// Mitsubishi GX Works2 project: TappingM6   PLC: FX1N/FX1NC

// global labels: Global1
VAR_GLOBAL
  XXFeed AT D52 : INT;
  XXRun AT M51 : BOOL;
  XXTarget AT D51 : INT;
  XXCurrent AT D50 : INT;
  XXArray AT D53 : ARRAY [0..5] OF INT;
  Foil3 AT M20 : BOOL;
  Foil4 AT M21 : BOOL;
  XXIMin AT X000 : BOOL;
  ZZIMin AT X001 : BOOL;
  ZZIMax AT X002 : BOOL;
  FoilExtractorIMax AT X003 : BOOL;
  XXODirection AT Y004 : BOOL;
  XXOPulse AT Y000 : BOOL;
  ZZOPulse AT Y001 : BOOL;
  RunStop AT M24 : BOOL;
  RunTest AT M23 : BOOL;
  FoilBlocker AT M54 : BOOL;
  FoilExtractor AT M55 : BOOL;
  RunState AT D20 : INT;
  Run AT M22 : BOOL;
  XXCurrentPulse AT D8140 : DINT;
  Foil3Array AT D200 : ARRAY [0..5] OF INT;
  Foil4Array AT D210 : ARRAY [0..5] OF INT;
  FoilIndex AT D70 : INT;
  RunIsTest AT M25 : BOOL;
  RunFeedXX AT D21 : INT;
  TestSensorFoil AT M30 : BOOL;
  FoilExtractorMin AT M31 : BOOL;
  FoilExtractorMax AT M32 : BOOL;
  FoilBlockerMin AT M33 : BOOL;
  FoilBlockerMax AT M34 : BOOL;
  RunStopEmergency AT M26 : BOOL;
  TestFoilTimeSeconds AT D23 : INT;
  MachineReady AT M27 : BOOL;
  Foil1Manual AT M28 : BOOL;
  Foil1ManualIRun AT X004 : BOOL;
  ZZCurrentPulse AT D8142 : DINT;
  ZZCurrent AT D60 : INT;
  ZZTarget AT D61 : INT;
  ZZFeed AT D62 : INT;
  ZZRun AT M61 : BOOL;
  RunFeedZZ AT D22 : INT;
  Foil3Offset AT D80 : INT;
  Foil4Offset AT D81 : INT;
  Foil1Offset AT D82 : INT;
  ZZDownPosition AT D83 : INT;
  ZZODirection AT Y005 : BOOL;
  AirOToggle AT Y006 : BOOL;
  Air AT M56 : BOOL;
  FoilBlockerOToggle AT Y003 : BOOL;
  FoilExtractorOToggle AT Y002 : BOOL;
  ZZDirection AT M60 : BOOL;
  XXDirection AT M50 : BOOL;
END_VAR

// task Task_01 (event TRUE, interval 0, priority 31): POU_01

PROGRAM POU_01
VAR
  fRise : BOOL;
  fFall : BOOL;
  fXXFeedPulse : INT;
  fFoilIndexLast : INT;
  fFoilChanged : BOOL;
  fTmp : BOOL;
  fArrayIndex : INT;
  fArrayIndexDouble : INT;
  fRunStart : BOOL;
  fArrayCount : INT;
  fGetOriginDone : BOOL;
  fStepReady : BOOL;
  fGetOrigin : BOOL;
  fFoilDone : BOOL;
  fFoilTimerEN : BOOL;
  fFoilExtractorTimerEN : BOOL;
  fZZFeedPulse : INT;
  fXXTarR : BOOL;
  fZZTarR : BOOL;
  fRunStateNext : BOOL;
  fFoilOffset : INT;
  fXXTarRTimerEN : BOOL;
  fZZTarRTimerEN : BOOL;
END_VAR
(*////////////////////////////////////////*)
(*  _____       _ _   _       _ _         *)
(* |_   _|     (_) | (_)     | (_)        *)
(*   | |  _ __  _| |_ _  __ _| |_ _______ *)
(*   | | | '_ \| | __| |/ _` | | |_  / _ \*)
(*  _| |_| | | | | |_| | (_| | | |/ /  __/*)
(* |_____|_| |_|_|\__|_|\__,_|_|_/___\___|*)
(*                                        *)
(*////////////////////////////////////////*)
DMOV(M8002, 10000, D8146);
MOV(M8002, 200, D8148);
MOV(M8002, 80, RunFeedXX);
MOV(M8002, 40, RunFeedZZ);
MOV(M8002, 170, Foil3Offset);
MOV(M8002, 170, Foil4Offset);
MOV(M8002, 11000, Foil1Offset);
MOV(M8002, 1200, ZZDownPosition);
MOV(M8002, 0, Foil3Array[0]); MOV(M8002, 3000, Foil3Array[1]); MOV(M8002, 6000, Foil3Array[2]);
MOV(M8002, 0, Foil4Array[0]); MOV(M8002, 2000, Foil4Array[1]); MOV(M8002, 4000, Foil4Array[2]); MOV(M8002, 6000, Foil4Array[3]);
RST(M8002, TestSensorFoil);
RST(M8002, MachineReady);
RST(M8002, FoilIndex);
RST(M8002, fFoilIndexLast);
MOV(M8002, 10, XXFeed);
MOV(M8002, 1, ZZFeed);
OUT_T(NOT MachineReady, TC0, 30);
SET(TC0, MachineReady);
(*////////////////////////////////////////////////////*)
(*  __  __       _                                    *)
(* |  \/  |     (_)                                   *)
(* | \  / | __ _ _ _ __    _ __ ___   ___ _ __  _   _ *)
(* | |\/| |/ _` | | '_ \  | '_ ` _ \ / _ \ '_ \| | | |*)
(* | |  | | (_| | | | | | | | | | | |  __/ | | | |_| |*)
(* |_|  |_|\__,_|_|_| |_| |_| |_| |_|\___|_| |_|\__,_|*)
(*                                                    *)
(*////////////////////////////////////////////////////*)
(*Foil selection*)
OUT(FoilIndex = 1, Foil1Manual);
OUT(FoilIndex = 3, Foil3);
OUT(FoilIndex = 4, Foil4);
SET(FoilIndex <> fFoilIndexLast, fFoilChanged);
SET(fFoilChanged AND NOT M100, fTmp); RST(fTmp, fFoilChanged); MOV(fTmp, fFoilIndexLast, FoilIndex); RST(fTmp, fTmp);
MOV(fFoilChanged, FoilIndex, fFoilIndexLast);
BMOV(fFoilChanged AND Foil3, D200, 3, D53);
MOV(fFoilChanged AND Foil3, 3, fArrayCount);
BMOV(fFoilChanged AND Foil4, D210, 4, D53);
MOV(fFoilChanged AND Foil4, 4, fArrayCount);
RST(fFoilChanged, fFoilChanged);
(*Run*)
PLS(Run, fRise); RST(fRise AND M100, RunIsTest); SET(fRise AND M100, fRunStart);
PLS(RunTest, fRise); SET(fRise AND M100, RunIsTest); SET(fRise AND M100, fRunStart);
MOV(fRunStart AND MachineReady AND (Foil3 OR Foil4 OR Foil1Manual), 1, RunState);
MOV(fRunStart AND Foil3, Foil3Offset, fFoilOffset);
MOV(fRunStart AND Foil4, Foil4Offset, fFoilOffset);
RST(fRunStart, fArrayIndexDouble);
RST(fRunStart, fRunStart);
(*Stop*)
PLS(RunStopEmergency, fRise); SET(fRise, fTmp);
RST(fTmp, XXRun);
RST(fTmp, ZZRun);
RST(fTmp, RunState);
RST(fTmp, FoilExtractor);
RST(fTmp, FoilBlocker);
RST(fTmp, fTmp);
(*|||||||||||||||||||||||||||||||||||||||||||||||||||||||||||||||||||||||||||||||||||||||||||||||||||||||||||||||||||||||||||||||||||||||||||||||||||||||||||*)
(*|||||||||||||||||||||||||||||||||||||||||||||||||||||||||||||||||||||||||||||||||||||||||||||||||||||||||||||||||||||||||||||||||||||||||||||||||||||||||||*)
INC(fRunStateNext, RunState); RST(fRunStateNext, fRunStateNext);
DECO(TRUE, RunState, 6, M100); (*From M100 to M163, this does not require fStepReady*)
DECO(TRUE, RunState, 6, M200); (*From M200 to M263, this require fStepReady*)
RST(fStepReady, fStepReady);
SET(fGetOrigin AND fXXTarR AND fZZTarR, fStepReady);
SET(fGetOriginDone AND fXXTarR AND fZZTarR AND NOT RunStop, fStepReady);
ZRST(NOT fStepReady, M200, M263);
(**)
SET(M101 AND fXXTarR AND fZZTarR, fTmp);
SET(fTmp, fGetOrigin);
RST(fTmp, fGetOriginDone);
MOV(fTmp, 10, RunState);
RST(fTmp, fTmp);
(*|||||||||||||||||||||||||||||||||||||||||||||||||||||||||||||||||||||||||||||||||||||||||||||||||||||||||||||||||||||||||||||||||||||||||||||||||||||||||||*)
(*|||||||||||||||||||||||||||||||||||||||||||||||||||||||||||||||||||||||||||||||||||||||||||||||||||||||||||||||||||||||||||||||||||||||||||||||||||||||||||*)
(*/////////////////////////////////////////////////////*)
(*   _____      _                      _       _       *)
(*  / ____|    | |                    (_)     (_)      *)
(* | |  __  ___| |_   ____   ___  _ __ _  __ _ _ _ __  *)
(* | | |_ |/ _ \ __| |_  /  / _ \| '__| |/ _` | | '_ \ *)
(* | |__| |  __/ |_   / /  | (_) | |  | | (_| | | | | |*)
(*  \_____|\___|\__| /___|  \___/|_|  |_|\__, |_|_| |_|*)
(*                                        __/ |        *)
(*                                       |___/         *)
(*/////////////////////////////////////////////////////*)
(*z at min, next*)
SET(M210 AND ZZIMin, fTmp);
RST(fTmp, ZZCurrentPulse);
SET(fTmp, fRunStateNext); RST(fTmp, fTmp);
(*z not at min, z up*)
SET(M210 AND NOT ZZIMin, fTmp);
RST(fTmp, ZZCurrentPulse); MOV(fTmp, -20000, ZZTarget); MOV(fTmp, 5, ZZFeed); SET(fTmp, ZZRun);
SET(fTmp, fRunStateNext); RST(fTmp, fTmp);
(*z up in min, z down*)
SET(M211, fTmp);
MOV(fTmp, 2000, ZZTarget); MOV(fTmp, 1, ZZFeed); SET(fTmp, ZZRun);
SET(fTmp, fRunStateNext); RST(fTmp, fTmp);
(*z down out min, z stop*)
SET(M112 AND NOT ZZIMin, fTmp);
RST(fTmp, ZZRun);
SET(fTmp, fRunStateNext); RST(fTmp, fTmp);
(*z down 0.5mm*)
SET(M213, fTmp);
RST(fTmp, ZZCurrentPulse); MOV(fTmp, 50, ZZTarget); MOV(fTmp, 1, ZZFeed); SET(fTmp, ZZRun);
SET(fTmp, fRunStateNext); RST(fTmp, fTmp);
(*z done*)
SET(M214, fTmp);
RST(fTmp, ZZCurrentPulse); RST(fTmp, ZZTarget); MOV(fTmp, RunFeedZZ, ZZFeed);
SET(fTmp, fRunStateNext); RST(fTmp, fTmp);
(*|||||||||||||||||||||||||||||||||||||||||||||||||||||||||||||||||||||||||||||||||||||||||||||||||||||||||||||||||||||||||||||||||||||||||||||||||||||||||||*)
(*|||||||||||||||||||||||||||||||||||||||||||||||||||||||||||||||||||||||||||||||||||||||||||||||||||||||||||||||||||||||||||||||||||||||||||||||||||||||||||*)
(*Get z origin -> Get x origin*)
SET(M215, fTmp);
MOV(fTmp, 20, RunState); RST(fTmp, fTmp);
(*//////////////////////////////////////////////////////*)
(*   _____      _                       _       _       *)
(*  / ____|    | |                     (_)     (_)      *)
(* | |  __  ___| |_  __  __   ___  _ __ _  __ _ _ _ __  *)
(* | | |_ |/ _ \ __| \ \/ /  / _ \| '__| |/ _` | | '_ \ *)
(* | |__| |  __/ |_   >  <  | (_) | |  | | (_| | | | | |*)
(*  \_____|\___|\__| /_/\_\  \___/|_|  |_|\__, |_|_| |_|*)
(*                                         __/ |        *)
(*                                        |___/         *)
(*//////////////////////////////////////////////////////*)
(*x at min, next*)
SET(M220 AND XXIMin, fTmp);
RST(fTmp, XXCurrentPulse);
SET(fTmp, fRunStateNext); RST(fTmp, fTmp);
(*x not at min, x back*)
SET(M220 AND NOT XXIMin, fTmp);
RST(fTmp, XXCurrentPulse); MOV(fTmp, -20000, XXTarget); MOV(fTmp, 10, XXFeed); SET(fTmp, XXRun);
SET(fTmp, fRunStateNext); RST(fTmp, fTmp);
(*x back in min, x forward*)
SET(M221, fTmp);
MOV(fTmp, 2000, XXTarget); MOV(fTmp, 1, XXFeed); SET(fTmp, XXRun);
SET(fTmp, fRunStateNext); RST(fTmp, fTmp);
(*x out min, x stop*)
SET(M122 AND NOT XXIMin, fTmp);
RST(fTmp, XXRun);
SET(fTmp, fRunStateNext); RST(fTmp, fTmp);
(*x forward 1mm*)
SET(M223, fTmp);
RST(fTmp, XXCurrentPulse); MOV(fTmp, 100, XXTarget); MOV(fTmp, 1, XXFeed); SET(fTmp, XXRun);
SET(fTmp, fRunStateNext); RST(fTmp, fTmp);
(*x done*)
SET(M224, fTmp);
RST(fTmp, XXCurrentPulse); RST(fTmp, XXTarget); MOV(fTmp, RunFeedXX, XXFeed);
MOV(fTmp AND NOT Foil1Manual, 25, RunState);
MOV(fTmp AND Foil1Manual, 50, RunState);
RST(fTmp, fGetOrigin);
SET(fTmp, fGetOriginDone);
RST(fTmp, fTmp);
(*/////////////////////////////////////////////////////*)
(*  _____                                  __      _ _ *)
(* |  __ \                                / _|    (_) |*)
(* | |__) | __ ___ _ __   __ _ _ __ ___  | |_ ___  _| |*)
(* |  ___/ '__/ _ \ '_ \ / _` | '__/ _ \ |  _/ _ \| | |*)
(* | |   | | |  __/ |_) | (_| | | |  __/ | || (_) | | |*)
(* |_|   |_|  \___| .__/ \__,_|_|  \___| |_| \___/|_|_|*)
(*                | |                                  *)
(*                |_|                                  *)
(*/////////////////////////////////////////////////////*)
(*Set initial position*)
SET(M225, fTmp);
RST(fTmp, FoilExtractor); SET(fTmp, FoilExtractorMin);
SET(fTmp, FoilBlocker);
SET(fTmp, fRunStateNext); RST(fTmp, fTmp);
(*Wait until meet*)
SET(M226 AND FoilExtractorMin AND FoilBlockerMax, fTmp);
SET(fTmp, fRunStateNext); RST(fTmp, fTmp);
(*|||||||||||||||||||||||||||||||||||||||||||||||||||||||||||||||||||||||||||||||||||||||||||||||||||||||||||||||||||||||||||||||||||||||||||||||||||||||||||*)
(*|||||||||||||||||||||||||||||||||||||||||||||||||||||||||||||||||||||||||||||||||||||||||||||||||||||||||||||||||||||||||||||||||||||||||||||||||||||||||||*)
(*Prepair foil -> Loop*)
SET(M227, fTmp);
MOV(fTmp, 30, RunState); RST(fTmp, fTmp);
(*//////////////////////////*)
(*  _                       *)
(* | |                      *)
(* | |     ___   ___  _ __  *)
(* | |    / _ \ / _ \| '_ \ *)
(* | |___| (_) | (_) | |_) |*)
(* |______\___/ \___/| .__/ *)
(*                   | |    *)
(*                   |_|    *)
(*//////////////////////////*)
(*set x*)
SET(M230, fTmp);
SET(fTmp, fFoilTimerEN);
OUT_T(fFoilTimerEN, TC184, 10000);
MOV(fTmp, fArrayIndexDouble MOD fArrayCount, fArrayIndex);
MOV(fTmp AND fArrayIndexDouble >= fArrayCount, fArrayCount - fArrayIndex - 1, fArrayIndex);
MOV(fTmp, XXArray[fArrayIndex] + fFoilOffset, XXTarget);
INC(fTmp, fArrayIndexDouble);
RST(fTmp AND fArrayIndexDouble = fArrayCount * 2, fArrayIndexDouble);
SET(fTmp, fRunStateNext); RST(fTmp, fTmp);
(*run x*)
SET(M231, fTmp);
SET(fTmp, XXRun);
SET(fTmp, fRunStateNext); RST(fTmp, fTmp);
(*run x done, run z down*)
SET(M232, fTmp);
MOV(fTmp, ZZDownPosition, ZZTarget); SET(fTmp, ZZRun);
SET(fTmp, fRunStateNext); RST(fTmp, fTmp);
(*run z down done, run z up*)
SET(M233, fTmp);
MOV(fTmp, 0, ZZTarget); SET(fTmp, ZZRun);
SET(fTmp, fRunStateNext); RST(fTmp, fTmp);
(*run z up done*)
SET(M234, fTmp);
RST(fTmp, fFoilDone);
SET(fTmp AND (fArrayIndexDouble = 0 OR fArrayIndexDouble = fArrayCount), fFoilDone);
MOV(fFoilDone, T184, TestFoilTimeSeconds);
RST(fFoilDone, fFoilTimerEN);
RST(fFoilDone, T184);
MOV(fTmp AND NOT fFoilDone, 30, RunState);
MOV(fTmp AND fFoilDone, 35, RunState);
RST(fTmp, fFoilDone);
RST(fTmp, fTmp);
(*blocker down*)
SET(M235, fTmp);
RST(fTmp, FoilBlocker);
SET(fTmp, fRunStateNext); RST(fTmp, fTmp);
(*blocker down done, extractor forward*)
SET(M236 AND FoilBlockerMin, fTmp);
SET(fTmp, FoilExtractor);
SET(fTmp, fRunStateNext); RST(fTmp, fTmp);
(*extractor forward done, blocker up*)
SET(M237 AND FoilExtractorMax, fTmp);
SET(fTmp, FoilBlocker);
SET(fTmp, Air);
SET(fTmp, fRunStateNext); RST(fTmp, fTmp);
(*blocker up done, extractor back*)
SET(M238 AND FoilBlockerMax, fTmp);
RST(fTmp, FoilExtractor);
SET(fTmp, fRunStateNext); RST(fTmp, fTmp);
(*extractor back done, return*)
SET(M239 AND FoilExtractorMin, fTmp);
MOV(fTmp AND RunIsTest, 0, RunState);
MOV(fTmp AND NOT RunIsTest, 30, RunState);
RST(fTmp, fTmp);
(*///////////////////////////////////*)
(*  __  __                         _ *)
(* |  \/  |                       | |*)
(* | \  / | __ _ _ __  _   _  __ _| |*)
(* | |\/| |/ _` | '_ \| | | |/ _` | |*)
(* | |  | | (_| | | | | |_| | (_| | |*)
(* |_|  |_|\__,_|_| |_|\__,_|\__,_|_|*)
(*                                   *)
(*///////////////////////////////////*)
(*set static x position*)
SET(M250, fTmp);
RST(fTmp, FoilExtractor);
RST(fTmp, FoilBlocker);
MOV(fTmp, Foil1Offset, XXTarget);
SET(fTmp, fRunStateNext); RST(fTmp, fTmp);
(*run x*)
SET(M251, fTmp);
SET(fTmp, XXRun);
SET(fTmp, fRunStateNext); RST(fTmp, fTmp);
(*run x done, run z down*)
PLS(Foil1ManualIRun, fRise);
SET(M252 AND fRise, fTmp);
MOV(fTmp, ZZDownPosition, ZZTarget); SET(fTmp, ZZRun);
SET(fTmp, fRunStateNext); RST(fTmp, fTmp);
(*run z down done, run z up*)
SET(M253, fTmp);
MOV(fTmp, 0, ZZTarget); SET(fTmp, ZZRun);
SET(fTmp, fRunStateNext); RST(fTmp, fTmp);
(*run z up done*)
SET(M254, fTmp);
MOV(fTmp, 52, RunState); RST(fTmp, fTmp);
(*|||||||||||||||||||||||||||||||||||||||||||||||||||||||||||||||||||||||||||||||||||||||||||||||||||||||||||||||||||||||||||||||||||||||||||||||||||||||||||*)
(*|||||||||||||||||||||||||||||||||||||||||||||||||||||||||||||||||||||||||||||||||||||||||||||||||||||||||||||||||||||||||||||||||||||||||||||||||||||||||||*)
PLS(M8012, fRise); MOV(fRise, DINT_TO_INT(XXCurrentPulse), XXCurrent); MOV(fRise, DINT_TO_INT(ZZCurrentPulse), ZZCurrent);
(**)
RST(XXRun, fXXTarR);
SET(XXRun AND XXTarget = DINT_TO_INT(XXCurrentPulse), fTmp); RST(fTmp, XXRun); RST(fTmp, fTmp);
PLS(XXRun, fRise); MOV(fRise, XXFeed * 100, fXXFeedPulse);
DRVA(XXRun, XXTarget, fXXFeedPulse, XXOPulse, XXODirection);
RST(M8029, XXRun);
OUT(XXODirection, XXDirection);
OUT(NOT XXRun AND NOT M8147, fXXTarRTimerEN); OUT_T(fXXTarRTimerEN, TC1, 1); SET(TC1, fXXTarR);
RST(NOT XXDirection AND XXIMin, XXRun);
(**)
(**)
RST(ZZRun, fZZTarR);
SET(ZZRun AND ZZTarget = DINT_TO_INT(ZZCurrentPulse), fTmp); RST(fTmp, ZZRun); RST(fTmp, fTmp);
PLS(ZZRun, fRise); MOV(fRise, ZZFeed * 100, fZZFeedPulse);
DRVA(ZZRun, ZZTarget, fZZFeedPulse, ZZOPulse, ZZODirection);
RST(M8029, ZZRun);
OUT(ZZODirection, ZZDirection);
OUT(NOT ZZRun AND NOT M8148, fZZTarRTimerEN); OUT_T(fZZTarRTimerEN, TC2, 1); SET(TC2, fZZTarR);
RST(NOT ZZDirection AND ZZIMin, ZZRun);
RST(ZZDirection AND ZZIMax, ZZRun);
(**)

OUT(FoilBlocker, FoilBlockerOToggle);
OUT(FoilExtractor, FoilExtractorOToggle);
OUT_T(Air, TC10, 2); RST(TC10, Air); OUT(Air, AirOToggle);
(**)
PLS(FoilExtractorMin, fRise); RST(fRise, FoilExtractorMax);
PLS(FoilExtractorMax, fRise); RST(fRise, FoilExtractorMin);
PLS(FoilBlockerMin, fRise); RST(fRise, FoilBlockerMax);
PLS(FoilBlockerMax, fRise); RST(fRise, FoilBlockerMin);
(**)
PLS(FoilExtractorIMax, fRise); SET(fRise, fFoilExtractorTimerEN);
OUT_T(NOT FoilExtractor AND fFoilExtractorTimerEN, TC11, 5); PLS(TC11, fRise); SET(fRise, FoilExtractorMin); RST(fRise, fFoilExtractorTimerEN);
SET(FoilExtractor AND fFoilExtractorTimerEN, FoilExtractorMax);
OUT_T(NOT FoilBlocker, TC12, 3); PLS(TC12, fRise); SET(fRise, FoilBlockerMin);
OUT_T(FoilBlocker, TC13, 3); PLS(TC13, fRise); SET(fRise, FoilBlockerMax);
END_PROGRAM
